// Brief: Master Arm Ready for Master Slave Control
FUNCTION_BLOCK PUBLIC FB_StateCtrlReady EXTENDS FB_MasterArmCtrlBase
VAR_INPUT
END_VAR
VAR_OUTPUT
END_VAR
VAR
END_VAR

METHOD PUBLIC init : BOOL
VAR_IN_OUT CONSTANT
	i_masterArm	:FB_MasterArm;
END_VAR
VAR_IN_OUT 
	r_masterArmCtrlCmd :ST_ArmCtrlCmds;
END_VAR

VAR
	j:INT;
	maxJntErr:LREAL;
	jntCtrlErr:Vec7d;
END_VAR
SUPER^.Init(i_masterArm,r_masterArmCtrlCmd);

// check if to hold the command joint position unchanged
checkToHoldLastCmds(i_masterArm,r_masterArmCtrlCmd);
END_METHOD

END_FUNCTION_BLOCK

(* stored: Version 1.1.0.1, ProductVersion 3.1.4024.12
   POU FB_StateCtrlReady: Id {b4863c0c-c549-4967-ab29-6a1152ef3cd8}, SpecialFunc None
   Method init: Id {2537cbc9-bbc0-4d20-a9bf-3a888748c955} *)
